ABB RobotStudio station: ABB_Simulatsioon1.rsstnx

Station ABB_Simulatsioon1 (saved by RobotStudio 25.1.11167.1)
Controller IRB1300_11_90, task T_ROB1: task frame (RAPID world) sits at (800, -100, 800) mm, rotated rx 0 ry 0 rz 180 deg in the station
Controller IRB1300_11_90
  mechanical unit ROB_1: IRB1300_11_90__01, 6 joints, base frame (0, 0, 0) mm
Layout (positions relative to the parent item):
  - IRB1300_11_90__01 [mechanism, from %ABB.RobotStudio.Models.IRB1300%\IRB1300_11_90__01.rslib] at (800, -100, 800) mm, rotated rx 0 ry 0 rz 180 deg; joint values [-0.4142, 0.4067, 0.3774, 2.5848, 0.8657, 0.3834] (rad or m)
  - SC_Konveier [smart component]
      signals: DI DI_ToodeKonveieril, DI DI_LiigutaToodet, DI DI_AnnaKruvi, DI DI_KinnitaKruvi1, DO DO_ToodeKeskel, DO DO_ToodeLõpus, DI DI_KinnitaKruvi2, DI DI_KinnitaKruvi3, DI DI_KinnitaKruvi4
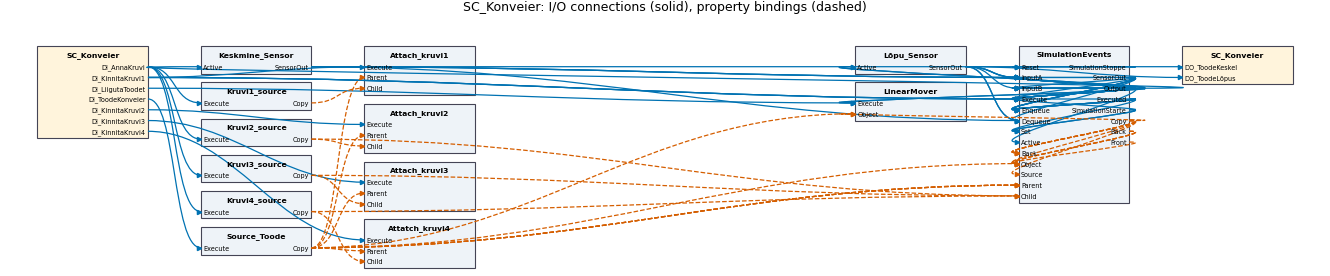
      connections:
        SimulationEvents.SimulationStopped -> LogicSRLatch.Reset
        PlaneSensor.SensorOut -> LogicGate.InputA
        LogicSRLatch.Output -> LogicGate_2.InputA
        LogicGate.Output -> LogicGate_2.InputB
        LogicGate_2.Output -> Source.Execute
        Source.Executed -> Queue.Enqueue
        PlaneSensor.SensorOut -> Queue.Dequeue
        SimulationEvents.SimulationStarted -> Hide.Execute
        Hide.Executed -> LogicSRLatch.Set
        PlaneSensor_2.SensorOut -> Queue_3.Enqueue
        PlaneSensor_2.SensorOut -> Queue_4.Enqueue
        PlaneSensor_2.SensorOut -> Queue_5.Enqueue
        LogicSRLatch.Output -> LogicGate_4.InputA
        PlaneSensor_4.SensorOut -> LogicGate_5.InputA
        LogicGate_5.Output -> LogicGate_4.InputB
        Source.Executed -> Queue_6.Enqueue
        PlaneSensor_4.SensorOut -> Queue_7.Enqueue
        PlaneSensor_4.SensorOut -> LinearMover.Execute
        PlaneSensor_4.SensorOut -> LogicGate_6.InputB
        LogicGate_6.Output -> LinearMover_4.Execute
        LogicGate_7.Output -> PlaneSensor.Active
        SimulationEvents.SimulationStarted -> LogicSRLatch_4.Set
        SimulationEvents.SimulationStopped -> LogicSRLatch_4.Reset
        LogicGate_8.Output -> Keskmine_Sensor.Active
        Keskmine_Sensor.SensorOut -> LogicGate_9.InputA
        LogicSRLatch_4.Output -> LogicGate_10.InputA
        LogicGate_9.Output -> LogicGate_10.InputB
        LogicGate_10.Output -> Source_6.Execute
        Source_6.Executed -> Queue_8.Enqueue
        LogicGate_11.Output -> Hide_2.Execute
        LogicGate_8.Output -> LogicGate_11.InputA
        LogicGate_8.Output -> Hide_3.Execute
        Source_6.Executed -> Hide_3.Execute
        LogicGate_14.Output -> Hide_5.Execute
        LogicGate_13.Output -> Hide_5.Execute
        Source_7.Executed -> Queue_10.Enqueue
        Lõpu_Sensor.SensorOut -> Queue_10.Dequeue
        SimulationEvents.SimulationStarted -> LogicSRLatch_5.Set
        SimulationEvents.SimulationStopped -> LogicSRLatch_5.Reset
        LogicSRLatch_5.Output -> LogicGate_15.InputA
        LogicGate_16.Output -> LogicGate_15.InputB
        Lõpu_Sensor.SensorOut -> LogicGate_16.InputA
        LogicGate_15.Output -> Source_8.Execute
        Source_8.Executed -> Queue_11.Enqueue
        Lõpu_Sensor.SensorOut -> Queue_11.Dequeue
        Keskmine_Sensor.SensorOut -> Queue_8.Dequeue
        Keskmine_Sensor.SensorOut -> LogicGate.InputA
        LogicGate.Output -> LogicGate_2.InputB
        Lõpu_Sensor.SensorOut -> LogicGate_3.InputA
        LogicGate_5.Output -> Lõpu_Sensor.Active
        LogicGate_2.Output -> LogicGate_4.InputA
        LogicGate_4.Output -> LinearMover.Execute
        Lõpu_Sensor.SensorOut -> LogicGate_4.InputB
        LogicGate_6.Output -> Lõpu_Sensor.Active
        Keskmine_Sensor.SensorOut -> LogicGate_7.InputA
        LogicGate_7.Output -> LogicGate_2.InputB
        LogicGate_2.Output -> LinearMover.Execute
        Lõpu_Sensor.SensorOut -> LogicGate_9.InputA
        LogicGate_9.Output -> LogicGate_8.InputB
        LogicGate_10.Output -> LogicGate_8.InputA
        LogicGate_8.Output -> LinearMover_14.Execute
        SC_Konveier.DI_AnnaKruvi -> Kruvi1_source.Execute
        SC_Konveier.DI_KinnitaKruvi1 -> Attach_kruvi1.Execute
        Keskmine_Sensor.SensorOut -> SC_Konveier.DO_ToodeKeskel
        Lõpu_Sensor.SensorOut -> SC_Konveier.DO_ToodeLõpus
        SC_Konveier.DI_LiigutaToodet -> LinearMover.Execute
        SC_Konveier.DI_ToodeKonveieril -> Source_Toode.Execute
        SC_Konveier.DI_KinnitaKruvi1 -> Attatch_kruvi2.Execute
        SC_Konveier.DI_KinnitaKruvi1 -> Attatch_kruvi3.Execute
        SC_Konveier.DI_KinnitaKruvi1 -> Attatch_kruvi4.Execute
        SC_Konveier.DI_AnnaKruvi -> Kruvi2_source.Execute
        SC_Konveier.DI_AnnaKruvi -> Kruvi3_source.Execute
        SC_Konveier.DI_AnnaKruvi -> Kruvi4_source.Execute
        SC_Konveier.DI_KinnitaKruvi2 -> Attach_kruvi2.Execute
        SC_Konveier.DI_KinnitaKruvi3 -> Attach_kruvi3.Execute
        SC_Konveier.DI_KinnitaKruvi4 -> Attatch_kruvi4.Execute
        Source.Copy => Queue_6.Back
        Source.Copy => Queue.Back
        Source_6.Copy => Hide_5.Object
        Source_6.Copy => Source_7.Source
        Source_7.Copy => Queue_10.Back
        Queue_8.Back => LinearMover2_3.Object
        Queue_8.Back => LinearMover_12.Object
        Source_9.Copy => LinearMover.Object
        Queue_8.Back => Sink.Object
        Queue_8.Front => LinearMover_11.Object
        Source_6.Copy => Queue_8.Back
        Source_Toode.Copy => LinearMover.Object
        Source_Toode.Copy => LinearMover_14.Object
        Source_Toode.Copy => Attacher_4.Parent
        Source_Toode.Copy => Attach_kruvi1.Parent
        Source_Toode.Copy => Attatch_kruvi3.Parent
        Source_Toode.Copy => Attatch_kruvi2.Parent
        Kruvi1_source.Copy => Attach_kruvi1.Child
        Kruvi2_source.Copy => Attatch_kruvi2.Child
        Source_Toode.Copy => Attatch_kruvi4.Parent
        Kruvi3_source.Copy => Attatch_kruvi3.Child
        Kruvi4_source.Copy => Attatch_kruvi4.Child
        Source_Toode.Copy => Attach_kruvi2.Parent
        Source_Toode.Copy => Attach_kruvi3.Parent
        Source_Toode.Copy => Attatch_kruvi4.Parent
        Kruvi2_source.Copy => Attach_kruvi2.Child
        Kruvi3_source.Copy => Attach_kruvi3.Child
        Kruvi4_source.Copy => Attatch_kruvi4.Child
    - Robot cell 3 [part] at (0, 0, 0) mm, rotated rx 90 ry 0 rz 0 deg, size 1635 x 2000 x 3000 mm
    - Toode R8 [part] at (0, 1100, 1009) mm, size 300 x 700 x 306 mm
    - Keskmine_Sensor [smart component, from Components\PlaneSensor.rslib]
        properties: Origin=[-0.2 -0.35 0.91]; Axis1=[0 0 0.1]; Axis2=[0.4 0 0]; Tag=(none); SenseMultiple=false; SensedPart=(none)
      - _sensorPart_ [part], size 400 x 0 x 100 mm
    - Lõpu_Sensor [smart component, from Components\PlaneSensor.rslib]
        properties: Origin=[-0.2 -1.4 0.91]; Axis1=[0 0 0.1]; Axis2=[0.4 0 0]; Tag=(none); SenseMultiple=false; SensedPart=(none)
      - _sensorPart_ [part], size 400 x 0 x 100 mm
    - LinearMover [smart component, from Components\LinearMover.rslib]
        properties: Object=(none); Direction=[0 -2.2 0]; Speed=0.5; Reference=Global; ReferenceObject=(none)
    - Source_Toode [smart component, from Components\Source.rslib] at (0, -3624, 0) mm
        properties: Source=Toode R8; Copy=(none); Parent=(none); Position=[0 1.1 1.009]; Orientation=[0 0 0]; Transient=false; PhysicsBehavior=-1
    - Kruvi3 [part] at (364.23, 281.68, 1142) mm, rotated rx 0 ry 90 rz 0 deg, size 6 x 5 x 5 mm
    - Kruvi3_source [smart component, from Components\Source.rslib]
        properties: Source=Kruvi3; Copy=(none); Parent=(none); Position=[0.364227 0.281681 1.145539]; Orientation=[0 1.5707963267949 0]; Transient=true; PhysicsBehavior=-1
    - Kruvi4_source [smart component, from Components\Source.rslib]
        properties: Source=Kruvi_4; Copy=(none); Parent=(none); Position=[0.364227 0.221681 1.145539]; Orientation=[0 1.5707963267949 0]; Transient=true; PhysicsBehavior=-1
    - Kruvi1_source [smart component, from Components\Source.rslib]
        properties: Source=Kruvi; Copy=(none); Parent=(none); Position=[0.364227 0.401681 1.145539]; Orientation=[0 1.5707963267949 0]; Transient=true; PhysicsBehavior=-1
    - Kruvi2_source [smart component, from Components\Source.rslib]
        properties: Source=Kruvi2; Copy=(none); Parent=(none); Position=[0.364227 0.341681 1.145539]; Orientation=[0 1.5707963267949 0]; Transient=true; PhysicsBehavior=-1
    - Kruvi2 [part] at (23.3, 178, 1149.93) mm, rotated rx 0 ry 90 rz 0 deg, size 6 x 5 x 5 mm
    - Kruvi [part] at (364.23, 401.68, 1146) mm, rotated rx 0 ry 90 rz 0 deg, size 6 x 5 x 5 mm
    - Kruvi_4 [part] at (364.23, 221.68, 1142) mm, rotated rx 0 ry 90 rz 0 deg, size 6 x 5 x 5 mm
    - Attach_kruvi1 [smart component, from Components\Attacher.rslib]
        properties: Parent=(none); Flange=0; Child=(none); Mount=false; Offset=[0 0 0]; Orientation=[0 0 0]
    - Attach_kruvi2 [smart component, from Components\Attacher.rslib]
        properties: Parent=(none); Flange=0; Child=(none); Mount=false; Offset=[0 0 0]; Orientation=[0 0 0]
    - Attach_kruvi3 [smart component, from Components\Attacher.rslib]
        properties: Parent=(none); Flange=0; Child=(none); Mount=false; Offset=[0 0 0]; Orientation=[0 0 0]
    - Attatch_kruvi4 [smart component, from Components\Attacher.rslib]
        properties: Parent=(none); Flange=0; Child=(none); Mount=false; Offset=[0 0 0]; Orientation=[0 0 0]
  - SC_Kruvikeeraja [smart component] at (209, 120.23, 1462.5) mm, rotated rx 0 ry -90 rz 0 deg
      signals: DI DI_Grip, DO DO_Attatch, DO DO_Detatch
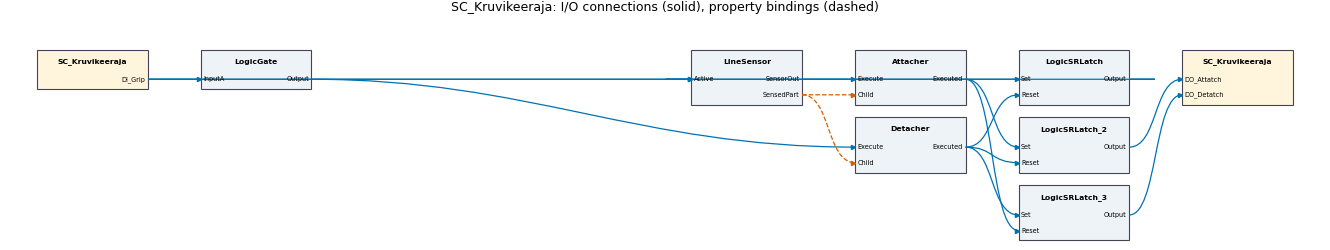
      connections:
        SC_Kruvikeeraja.DI_Grip -> LogicSRLatch.Set
        LineSensor.SensorOut -> Attacher.Execute
        Attacher.Executed -> LogicSRLatch_2.Set
        LogicSRLatch_2.Output -> SC_Kruvikeeraja.DO_Attatch
        SC_Kruvikeeraja.DI_Grip -> LogicGate.InputA
        LogicGate.Output -> Detacher.Execute
        Detacher.Executed -> LogicSRLatch_3.Set
        LogicSRLatch_3.Output -> SC_Kruvikeeraja.DO_Detatch
        Detacher.Executed -> LogicSRLatch.Reset
        Attacher.Executed -> LogicSRLatch_3.Reset
        Detacher.Executed -> LogicSRLatch_2.Reset
        LogicSRLatch.Output -> LineSensor.Active
        SC_Kruvikeeraja.DI_Grip -> LineSensor.Active
        LineSensor.SensedPart => Attacher.Child
        LineSensor.SensedPart => Detacher.Child
    - LineSensor [smart component, from Components\LineSensor.rslib]
        properties: Start=[-0.338500012541908 -0.000751017155122269 0.119996990466194]; End=[-0.342063902559134 -0.000723018135234478 0.119996990353048]; Length=0.003564; Radius=0.001; Tag=(none); SenseMultiple=false; SensedPart=(none); SensedPoint=[0.0889999923706055 0.119481979370117 1.101]
      - _sensorPart_ [part], size 3.6 x 2 x 2 mm
    - Attacher [smart component, from Components\Attacher.rslib]
        properties: Parent=KruvikeerajaABB_V2; Flange=0; Child=(none); Mount=false; Offset=[0 0 0]; Orientation=[0 0 0]
    - LogicSRLatch_2 [smart component, from Components\LogicSRLatch.rslib]
    - LogicGate [smart component, from Components\LogicGate.rslib]
        properties: Operator=NOT; Delay=0.5
    - Detacher [smart component, from Components\Detacher.rslib]
        properties: Child=(none); KeepPosition=true
    - LogicSRLatch_3 [smart component, from Components\LogicSRLatch.rslib]
    - KruvikeerajaABB_V2 [mechanism] at (0, 0, 0) mm
        TCP TCP_KruvikeerajaABB_V2 at (-636.74, -16.02, 73.26) mm, rotated rx -90 ry -74 rz 90 deg
        links: Tool
Attachment: SC_Kruvikeeraja is attached to IRB1300_11_90__01 / Link6
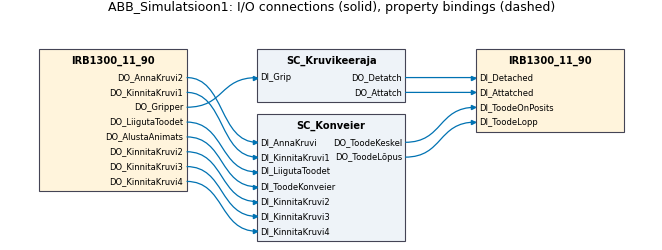
Station logic (signal -> signal, property => property):
  IRB1300_11_90.DO_AnnaKruvi2 -> SC_Konveier.DI_AnnaKruvi
  IRB1300_11_90.DO_KinnitaKruvi1 -> SC_Konveier.DI_KinnitaKruvi1
  IRB1300_11_90.DO_Gripper -> SC_Kruvikeeraja.DI_Grip
  SC_Kruvikeeraja.DO_Detatch -> IRB1300_11_90.DI_Detached
  SC_Kruvikeeraja.DO_Attatch -> IRB1300_11_90.DI_Attatched
  SC_Konveier.DO_ToodeKeskel -> IRB1300_11_90.DI_ToodeOnPositsioonil
  IRB1300_11_90.DO_LiigutaToodet -> SC_Konveier.DI_LiigutaToodet
  SC_Konveier.DO_ToodeLõpus -> IRB1300_11_90.DI_ToodeLopp
  IRB1300_11_90.DO_AlustaAnimatsioon -> SC_Konveier.DI_ToodeKonveieril
  IRB1300_11_90.DO_KinnitaKruvi2 -> SC_Konveier.DI_KinnitaKruvi2
  IRB1300_11_90.DO_KinnitaKruvi3 -> SC_Konveier.DI_KinnitaKruvi3
  IRB1300_11_90.DO_KinnitaKruvi4 -> SC_Konveier.DI_KinnitaKruvi4
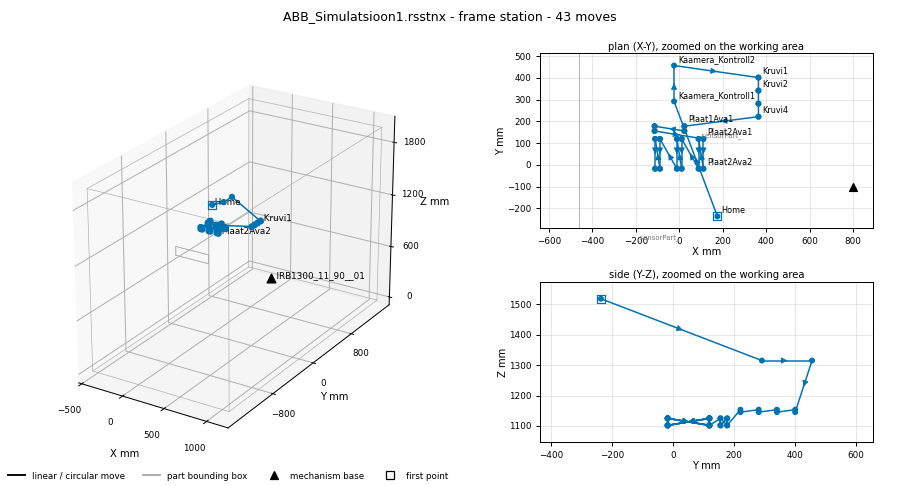
[picture p0: tool path of ABB_Simulatsioon1.rsstnx in frame station, 43 of 43 moves have a stored position in this frame; points joined in program order, loops and branches not executed]
Targets, tools, work objects and paths stored in the station, written as RAPID:
! task T_ROB1
MODULE CalibData
  PERS tooldata TCP_KruvikeerajaABB_V2:=[TRUE,[[-337.5,-0.733,119.997],[0.707106781,0,-0.707106781,0]],[1,[0,0,1],[1,0,0,0],0,0,0]];
ENDMODULE

! task T_ROB1
MODULE Module1
  CONST robtarget Kruvi1:=[[435.773415754,-501.680709441,345.539232334],[0,1,0,0],[-1,1,0,0],[9E+09,9E+09,9E+09,9E+09,9E+09,9E+09]];
  CONST robtarget Kruvi2:=[[435.773,-441.681,345.539],[0,1,0,0],[-1,1,0,0],[9E+09,9E+09,9E+09,9E+09,9E+09,9E+09]];
  CONST robtarget Kruvi3:=[[435.773,-381.681,345.539],[0,1,0,0],[-1,1,0,0],[9E+09,9E+09,9E+09,9E+09,9E+09,9E+09]];
  CONST robtarget Kruvi4:=[[435.773,-321.681,345.539],[0,1,0,0],[-1,1,0,0],[9E+09,9E+09,9E+09,9E+09,9E+09,9E+09]];
  CONST robtarget Kruvi1Kohal:=[[435.773462693,-501.680676163,353.539305771],[0.000000048,1,-0.000000288,0.000000324],[-1,1,0,0],[9E+09,9E+09,9E+09,9E+09,9E+09,9E+09]];
  CONST robtarget Kruvi2Kohal:=[[435.7699882,-441.680010312,353.539989026],[-0.000000023,1,-0.000000024,0.000000018],[-1,1,0,0],[9E+09,9E+09,9E+09,9E+09,9E+09,9E+09]];
  CONST robtarget Kruvi3Kohal:=[[435.769987813,-381.67998072,353.539970582],[-0.000000018,1,0.000000005,-0.000000012],[-1,1,0,0],[9E+09,9E+09,9E+09,9E+09,9E+09,9E+09]];
  CONST robtarget Kruvi4Kohal:=[[435.769991737,-321.679984075,353.539981013],[0.000000016,1,0.00000006,-0.000000014],[-1,1,0,0],[9E+09,9E+09,9E+09,9E+09,9E+09,9E+09]];
  CONST robtarget Plaat1Ava1:=[[776.7,-278,302],[0,1,0,0],[-1,1,0,0],[9E+09,9E+09,9E+09,9E+09,9E+09,9E+09]];
  CONST robtarget Plaat1Ava2:=[[776.7,-256,302],[0,1,0,0],[-1,1,0,0],[9E+09,9E+09,9E+09,9E+09,9E+09,9E+09]];
  CONST robtarget Plaat1Ava3:=[[913.7,-278,302],[0,1,0,0],[-1,1,0,0],[9E+09,9E+09,9E+09,9E+09,9E+09,9E+09]];
  CONST robtarget Plaat1Ava4:=[[913.7,-256,302],[0,1,0,0],[-1,1,0,0],[9E+09,9E+09,9E+09,9E+09,9E+09,9E+09]];
  CONST robtarget Plaat2Ava1:=[[689,-219.5,302],[0,1,0,0],[-1,1,0,0],[9E+09,9E+09,9E+09,9E+09,9E+09,9E+09]];
  CONST robtarget Plaat2Ava3:=[[711,-219.5,302],[0,1,0,0],[-1,1,0,0],[9E+09,9E+09,9E+09,9E+09,9E+09,9E+09]];
  CONST robtarget Plaat2Ava2:=[[689,-82.5,302],[0,1,0,0],[-1,1,0,0],[9E+09,9E+09,9E+09,9E+09,9E+09,9E+09]];
  CONST robtarget Plaat2Ava4:=[[711,-82.5,302.3],[0,1,0,0],[-1,1,0,0],[9E+09,9E+09,9E+09,9E+09,9E+09,9E+09]];
  CONST robtarget Plaat3Ava1:=[[789,-219.5,302.3],[0,1,0,0],[-1,1,0,0],[9E+09,9E+09,9E+09,9E+09,9E+09,9E+09]];
  CONST robtarget Plaat3Ava3:=[[811,-219.5,302],[0,1,0,0],[-1,1,0,0],[9E+09,9E+09,9E+09,9E+09,9E+09,9E+09]];
  CONST robtarget Plaat3Ava2:=[[789,-82.5,302],[0,1,0,0],[-1,1,0,0],[9E+09,9E+09,9E+09,9E+09,9E+09,9E+09]];
  CONST robtarget Plaat3Ava4:=[[811,-82.5,302],[0,1,0,0],[-1,1,0,0],[9E+09,9E+09,9E+09,9E+09,9E+09,9E+09]];
  CONST robtarget Plaat4Ava1:=[[889,-219.5,302],[0,1,0,0],[-1,1,0,0],[9E+09,9E+09,9E+09,9E+09,9E+09,9E+09]];
  CONST robtarget Plaat4Ava3:=[[911,-219.5,302],[0,1,0,0],[-1,1,0,0],[9E+09,9E+09,9E+09,9E+09,9E+09,9E+09]];
  CONST robtarget Plaat4Ava2:=[[889,-82.5,302],[0,1,0,0],[-1,1,0,0],[9E+09,9E+09,9E+09,9E+09,9E+09,9E+09]];
  CONST robtarget Plaat4Ava4:=[[911,-82.5,302],[0,1,0,0],[-1,1,0,0],[9E+09,9E+09,9E+09,9E+09,9E+09,9E+09]];
  CONST robtarget Plaat1Ava1Kohal:=[[776.699988596,-278.000008446,324.99997644],[0.000000006,1,-0.000000012,-0.000000015],[-1,1,0,0],[9E+09,9E+09,9E+09,9E+09,9E+09,9E+09]];
  CONST robtarget Plaat1Ava2Kohal:=[[776.700008221,-255.999999816,324.999992221],[-0.000000033,1,-0.000000036,0.000000011],[-1,1,0,0],[9E+09,9E+09,9E+09,9E+09,9E+09,9E+09]];
  CONST robtarget Plaat1Ava3Kohal:=[[913.699949436,-278.000016466,325.000003515],[0.000000045,1,0.000000018,-0.000000009],[-1,1,0,0],[9E+09,9E+09,9E+09,9E+09,9E+09,9E+09]];
  CONST robtarget Plaat1Ava4Kohal:=[[913.699959848,-256.000000869,324.999974095],[-0.000000001,1,0.000000016,-0.000000006],[-1,1,0,0],[9E+09,9E+09,9E+09,9E+09,9E+09,9E+09]];
  CONST robtarget Plaat2Ava1Kohal:=[[689.00000639,-219.499994539,324.999995823],[-0.000000032,1,-0.000000037,0.000000009],[-1,1,0,0],[9E+09,9E+09,9E+09,9E+09,9E+09,9E+09]];
  CONST robtarget Plaat2Ava2Kohal:=[[688.999990388,-82.500005343,324.999986755],[0.000000005,1,0.000000004,-0.000000001],[-1,1,0,0],[9E+09,9E+09,9E+09,9E+09,9E+09,9E+09]];
  CONST robtarget Plaat2Ava3Kohal:=[[711.000015543,-219.500016054,325.000003962],[0.000000018,1,0.000000009,0.000000011],[-1,1,0,0],[9E+09,9E+09,9E+09,9E+09,9E+09,9E+09]];
  CONST robtarget Plaat2Ava4Kohal:=[[711.000006872,-82.499995857,324.999991213],[-0.000000017,1,-0.000000018,-0.000000007],[-1,1,0,0],[9E+09,9E+09,9E+09,9E+09,9E+09,9E+09]];
  CONST robtarget Plaat3Ava1Kohal:=[[788.999954385,-219.500007427,324.999989863],[-0.000000007,1,-0.000000018,-0.000000001],[-1,1,0,0],[9E+09,9E+09,9E+09,9E+09,9E+09,9E+09]];
  CONST robtarget Plaat3Ava2Kohal:=[[788.999960308,-82.500019594,324.999989448],[0.000000038,1,0.000000031,0.000000002],[-1,1,0,0],[9E+09,9E+09,9E+09,9E+09,9E+09,9E+09]];
  CONST robtarget Plaat3Ava3Kohal:=[[810.999956974,-219.49999925,324.999974055],[0,1,0,-0.000000021],[-1,1,0,0],[9E+09,9E+09,9E+09,9E+09,9E+09,9E+09]];
  CONST robtarget Plaat3Ava4Kohal:=[[810.999978006,-82.499999129,324.999991294],[-0.000000014,1,-0.00000001,0.000000008],[-1,1,0,0],[9E+09,9E+09,9E+09,9E+09,9E+09,9E+09]];
  CONST robtarget Plaat4Ava1Kohal:=[[888.999969588,-219.500011208,325.000002169],[0.000000027,1,0.000000013,-0.000000009],[-1,1,0,0],[9E+09,9E+09,9E+09,9E+09,9E+09,9E+09]];
  CONST robtarget Plaat4Ava2Kohal:=[[888.999978236,-82.500004985,325.000008624],[0.00000001,1,0.000000004,0.000000004],[-1,1,0,0],[9E+09,9E+09,9E+09,9E+09,9E+09,9E+09]];
  CONST robtarget Plaat4Ava3Kohal:=[[911.000006802,-219.500006563,325.000022867],[-0.000000006,1,-0.000000006,0.000000026],[-1,1,0,0],[9E+09,9E+09,9E+09,9E+09,9E+09,9E+09]];
  CONST robtarget Plaat4Ava4Kohal:=[[910.999983403,-82.499984451,324.99998112],[-0.000000039,1,-0.000000025,-0.000000012],[-1,1,0,0],[9E+09,9E+09,9E+09,9E+09,9E+09,9E+09]];
  CONST robtarget Home:=[[624.438234891,136.898577549,718.16254704],[0.083448839,0.853960657,0.500049797,0.11720788],[-1,1,0,0],[9E+09,9E+09,9E+09,9E+09,9E+09,9E+09]];
  CONST robtarget Kaamera_Kontroll1:=[[823.999822834,-392.149885078,515.115078467],[0.500000077,0.866025359,-0.000000271,-0.000000033],[-1,1,-1,0],[9E+09,9E+09,9E+09,9E+09,9E+09,9E+09]];
  CONST robtarget Kaamera_Kontroll2:=[[823.99956152,-557.150115019,515.115372568],[0.500000401,0.866025172,-0.000000055,-0.000000089],[-1,1,-1,0],[9E+09,9E+09,9E+09,9E+09,9E+09,9E+09]];
  PROC Path_10()
    MoveL Home,v500,fine,TCP_KruvikeerajaABB_V2\WObj:=wobj0;
    MoveL Kaamera_Kontroll1,v500,fine,TCP_KruvikeerajaABB_V2\WObj:=wobj0;
    MoveL Kaamera_Kontroll2,v500,fine,TCP_KruvikeerajaABB_V2\WObj:=wobj0;
    MoveL Kruvi1,v500,fine,TCP_KruvikeerajaABB_V2\WObj:=wobj0;
    MoveL Kruvi1Kohal,v500,fine,TCP_KruvikeerajaABB_V2\WObj:=wobj0;
    MoveL Kruvi2,v500,fine,TCP_KruvikeerajaABB_V2\WObj:=wobj0;
    MoveL Kruvi2Kohal,v500,fine,TCP_KruvikeerajaABB_V2\WObj:=wobj0;
    MoveL Kruvi3,v500,fine,TCP_KruvikeerajaABB_V2\WObj:=wobj0;
    MoveL Kruvi3Kohal,v500,fine,TCP_KruvikeerajaABB_V2\WObj:=wobj0;
    MoveL Kruvi4,v500,fine,TCP_KruvikeerajaABB_V2\WObj:=wobj0;
    MoveL Kruvi4Kohal,v500,fine,TCP_KruvikeerajaABB_V2\WObj:=wobj0;
    MoveL Plaat1Ava1,v500,fine,TCP_KruvikeerajaABB_V2\WObj:=wobj0;
    MoveL Plaat1Ava1Kohal,v500,fine,TCP_KruvikeerajaABB_V2\WObj:=wobj0;
    MoveL Plaat1Ava2,v500,fine,TCP_KruvikeerajaABB_V2\WObj:=wobj0;
    MoveL Plaat1Ava2Kohal,v500,fine,TCP_KruvikeerajaABB_V2\WObj:=wobj0;
    MoveL Plaat1Ava3,v500,fine,TCP_KruvikeerajaABB_V2\WObj:=wobj0;
    MoveL Plaat1Ava3Kohal,v500,fine,TCP_KruvikeerajaABB_V2\WObj:=wobj0;
    MoveL Plaat1Ava4,v500,fine,TCP_KruvikeerajaABB_V2\WObj:=wobj0;
    MoveL Plaat1Ava4Kohal,v500,fine,TCP_KruvikeerajaABB_V2\WObj:=wobj0;
    MoveL Plaat2Ava1,v500,fine,TCP_KruvikeerajaABB_V2\WObj:=wobj0;
    MoveL Plaat2Ava1Kohal,v500,fine,TCP_KruvikeerajaABB_V2\WObj:=wobj0;
    MoveL Plaat2Ava2,v500,fine,TCP_KruvikeerajaABB_V2\WObj:=wobj0;
    MoveL Plaat2Ava2Kohal,v500,fine,TCP_KruvikeerajaABB_V2\WObj:=wobj0;
    MoveL Plaat2Ava3,v500,fine,TCP_KruvikeerajaABB_V2\WObj:=wobj0;
    MoveL Plaat2Ava3Kohal,v500,fine,TCP_KruvikeerajaABB_V2\WObj:=wobj0;
    MoveL Plaat2Ava4,v500,fine,TCP_KruvikeerajaABB_V2\WObj:=wobj0;
    MoveL Plaat2Ava4Kohal,v500,fine,TCP_KruvikeerajaABB_V2\WObj:=wobj0;
    MoveL Plaat3Ava1,v500,fine,TCP_KruvikeerajaABB_V2\WObj:=wobj0;
    MoveL Plaat3Ava1Kohal,v500,fine,TCP_KruvikeerajaABB_V2\WObj:=wobj0;
    MoveL Plaat3Ava2,v500,fine,TCP_KruvikeerajaABB_V2\WObj:=wobj0;
    MoveL Plaat3Ava2Kohal,v500,fine,TCP_KruvikeerajaABB_V2\WObj:=wobj0;
    MoveL Plaat3Ava3,v500,fine,TCP_KruvikeerajaABB_V2\WObj:=wobj0;
    MoveL Plaat3Ava3Kohal,v500,fine,TCP_KruvikeerajaABB_V2\WObj:=wobj0;
    MoveL Plaat3Ava4,v500,fine,TCP_KruvikeerajaABB_V2\WObj:=wobj0;
    MoveL Plaat3Ava4Kohal,v500,fine,TCP_KruvikeerajaABB_V2\WObj:=wobj0;
    MoveL Plaat4Ava1,v500,fine,TCP_KruvikeerajaABB_V2\WObj:=wobj0;
    MoveL Plaat4Ava1Kohal,v500,fine,TCP_KruvikeerajaABB_V2\WObj:=wobj0;
    MoveL Plaat4Ava2,v500,fine,TCP_KruvikeerajaABB_V2\WObj:=wobj0;
    MoveL Plaat4Ava2Kohal,v500,fine,TCP_KruvikeerajaABB_V2\WObj:=wobj0;
    MoveL Plaat4Ava3,v500,fine,TCP_KruvikeerajaABB_V2\WObj:=wobj0;
    MoveL Plaat4Ava3Kohal,v500,fine,TCP_KruvikeerajaABB_V2\WObj:=wobj0;
    MoveL Plaat4Ava4,v500,fine,TCP_KruvikeerajaABB_V2\WObj:=wobj0;
    MoveL Plaat4Ava4Kohal,v500,fine,TCP_KruvikeerajaABB_V2\WObj:=wobj0;
  ENDPROC
ENDMODULE

